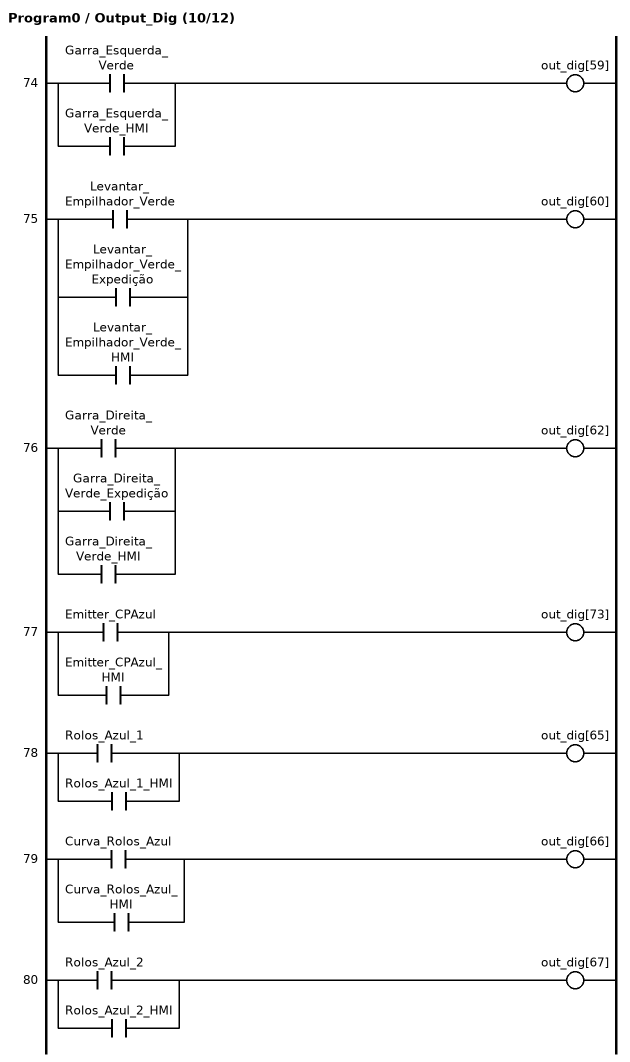
(* [picture p24: Program0 / Output_Dig, rungs 74-80] *)
(* Rung 74 *)
out_dig[59] := Garra_Esquerda_Verde OR Garra_Esquerda_Verde_HMI;
(* Rung 75 *)
out_dig[60] := Levantar_Empilhador_Verde OR Levantar_Empilhador_Verde_Expedição OR Levantar_Empilhador_Verde_HMI;
(* Rung 76 *)
out_dig[62] := Garra_Direita_Verde OR Garra_Direita_Verde_Expedição OR Garra_Direita_Verde_HMI;
(* Rung 77 *)
out_dig[73] := Emitter_CPAzul OR Emitter_CPAzul_HMI;
(* Rung 78 *)
out_dig[65] := Rolos_Azul_1 OR Rolos_Azul_1_HMI;
(* Rung 79 *)
out_dig[66] := Curva_Rolos_Azul OR Curva_Rolos_Azul_HMI;
(* Rung 80 *)
out_dig[67] := Rolos_Azul_2 OR Rolos_Azul_2_HMI;

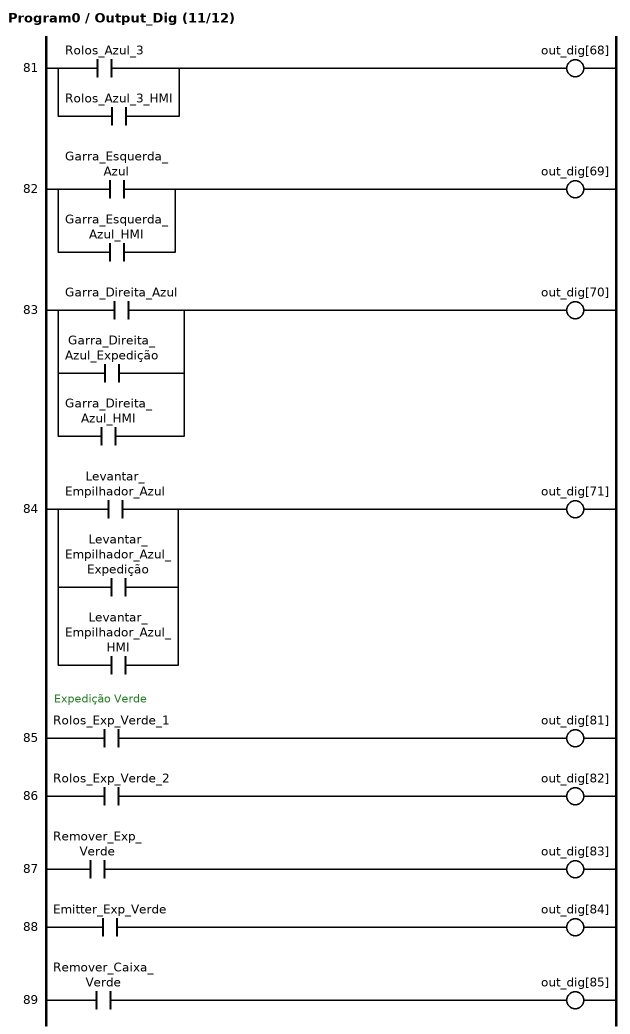
(* Rung 81 *)
out_dig[68] := Rolos_Azul_3 OR Rolos_Azul_3_HMI;
(* Rung 82 *)
out_dig[69] := Garra_Esquerda_Azul OR Garra_Esquerda_Azul_HMI;
(* Rung 83 *)
out_dig[70] := Garra_Direita_Azul OR Garra_Direita_Azul_Expedição OR Garra_Direita_Azul_HMI;
(* Rung 84 *)
out_dig[71] := Levantar_Empilhador_Azul OR Levantar_Empilhador_Azul_Expedição OR Levantar_Empilhador_Azul_HMI;
(* Rung 85: Expedição Verde *)
out_dig[81] := Rolos_Exp_Verde_1;
(* Rung 86 *)
out_dig[82] := Rolos_Exp_Verde_2;
(* Rung 87 *)
out_dig[83] := Remover_Exp_Verde;
(* Rung 88 *)
out_dig[84] := Emitter_Exp_Verde;
(* Rung 89 *)
out_dig[85] := Remover_Caixa_Verde;

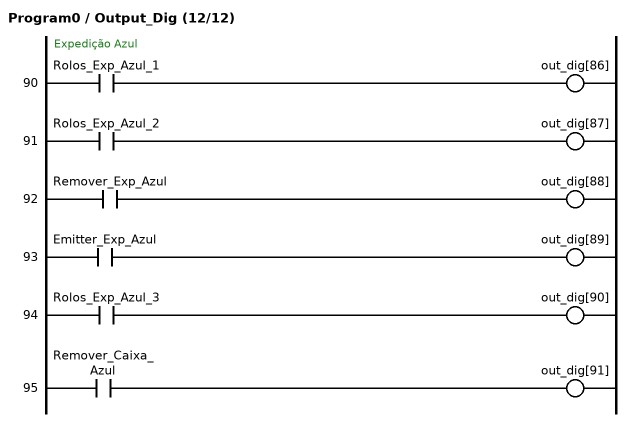
(* Rung 90: Expedição Azul *)
out_dig[86] := Rolos_Exp_Azul_1;
(* Rung 91 *)
out_dig[87] := Rolos_Exp_Azul_2;
(* Rung 92 *)
out_dig[88] := Remover_Exp_Azul;
(* Rung 93 *)
out_dig[89] := Emitter_Exp_Azul;
(* Rung 94 *)
out_dig[90] := Rolos_Exp_Azul_3;
(* Rung 95 *)
out_dig[91] := Remover_Caixa_Azul;

(* Section Separação_Inicial_Etapas: ladder, written here as Structured Text *)

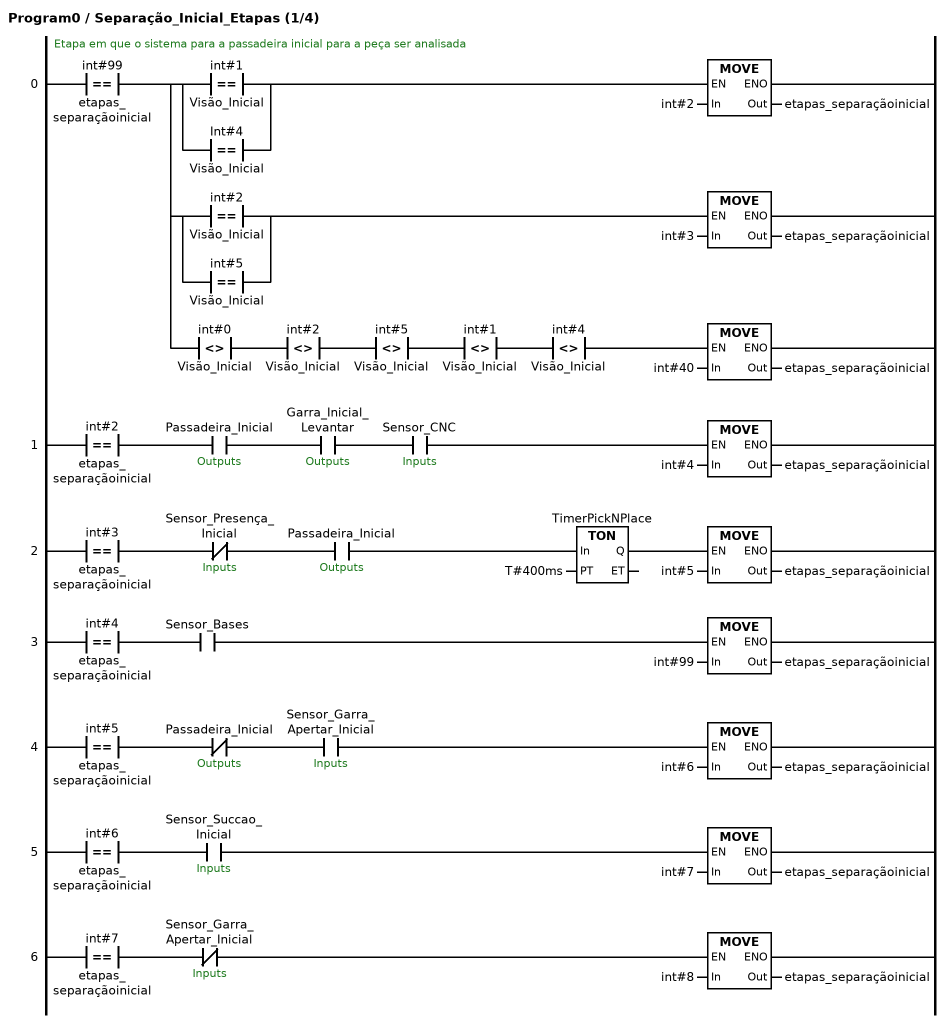
(* Rung 0: Etapa em que o sistema para a passadeira inicial para a peça ser analisada *)
_p4 := int#99 = etapas_separaçãoinicial;
IF (int#99 = etapas_separaçãoinicial) AND ((int#1 = Visão_Inicial) OR (Int#4 = Visão_Inicial)) THEN
    etapas_separaçãoinicial := int#2;
END_IF;
IF _p4 AND ((int#2 = Visão_Inicial) OR (int#5 = Visão_Inicial)) THEN
    etapas_separaçãoinicial := int#3;
END_IF;
IF _p4 AND (int#0 <> Visão_Inicial) AND (int#2 <> Visão_Inicial) AND (int#5 <> Visão_Inicial) AND (int#1 <> Visão_Inicial) AND (int#4 <> Visão_Inicial) THEN
    etapas_separaçãoinicial := int#40;
END_IF;
(* Rung 1 *)
IF (int#2 = etapas_separaçãoinicial) AND Passadeira_Inicial AND Garra_Inicial_Levantar AND Sensor_CNC THEN
    etapas_separaçãoinicial := int#4;
END_IF;
(* Rung 2 *)
TimerPickNPlace(In := (int#3 = etapas_separaçãoinicial) AND NOT Sensor_Presença_Inicial AND Passadeira_Inicial, PT := T#400ms);
IF TimerPickNPlace.Q THEN etapas_separaçãoinicial := int#5; END_IF;
(* Rung 3 *)
IF (int#4 = etapas_separaçãoinicial) AND Sensor_Bases THEN etapas_separaçãoinicial := int#99; END_IF;
(* Rung 4 *)
IF (int#5 = etapas_separaçãoinicial) AND NOT Passadeira_Inicial AND Sensor_Garra_Apertar_Inicial THEN
    etapas_separaçãoinicial := int#6;
END_IF;
(* Rung 5 *)
IF (int#6 = etapas_separaçãoinicial) AND Sensor_Succao_Inicial THEN
    etapas_separaçãoinicial := int#7;
END_IF;
(* Rung 6 *)
IF (int#7 = etapas_separaçãoinicial) AND NOT Sensor_Garra_Apertar_Inicial THEN
    etapas_separaçãoinicial := int#8;
END_IF;

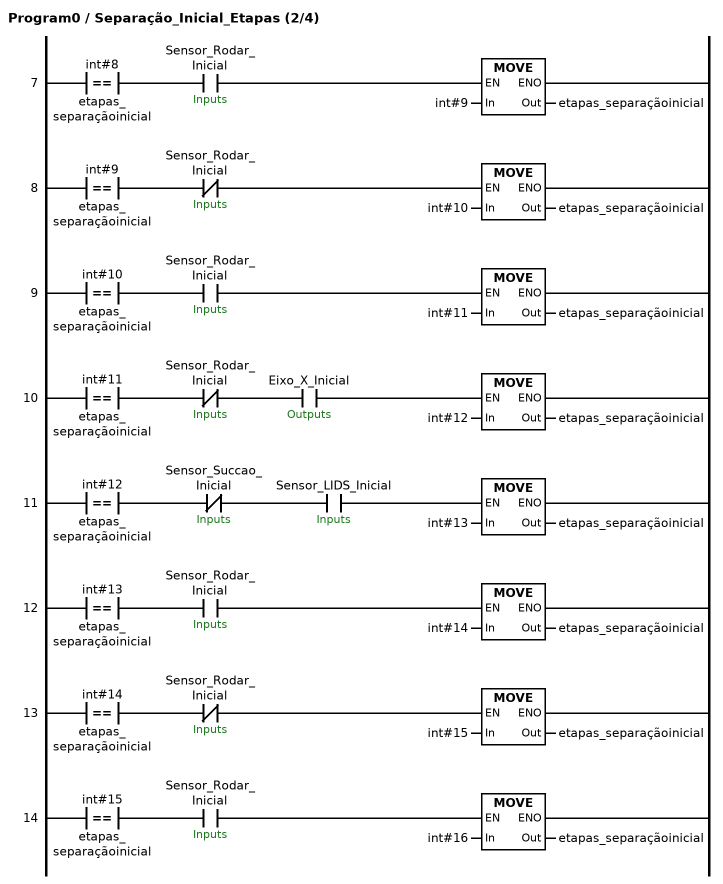
(* Rung 7 *)
IF (int#8 = etapas_separaçãoinicial) AND Sensor_Rodar_Inicial THEN
    etapas_separaçãoinicial := int#9;
END_IF;
(* Rung 8 *)
IF (int#9 = etapas_separaçãoinicial) AND NOT Sensor_Rodar_Inicial THEN
    etapas_separaçãoinicial := int#10;
END_IF;
(* Rung 9 *)
IF (int#10 = etapas_separaçãoinicial) AND Sensor_Rodar_Inicial THEN
    etapas_separaçãoinicial := int#11;
END_IF;
(* Rung 10 *)
IF (int#11 = etapas_separaçãoinicial) AND NOT Sensor_Rodar_Inicial AND Eixo_X_Inicial THEN
    etapas_separaçãoinicial := int#12;
END_IF;
(* Rung 11 *)
IF (int#12 = etapas_separaçãoinicial) AND NOT Sensor_Succao_Inicial AND Sensor_LIDS_Inicial THEN
    etapas_separaçãoinicial := int#13;
END_IF;
(* Rung 12 *)
IF (int#13 = etapas_separaçãoinicial) AND Sensor_Rodar_Inicial THEN
    etapas_separaçãoinicial := int#14;
END_IF;
(* Rung 13 *)
IF (int#14 = etapas_separaçãoinicial) AND NOT Sensor_Rodar_Inicial THEN
    etapas_separaçãoinicial := int#15;
END_IF;
(* Rung 14 *)
IF (int#15 = etapas_separaçãoinicial) AND Sensor_Rodar_Inicial THEN
    etapas_separaçãoinicial := int#16;
END_IF;

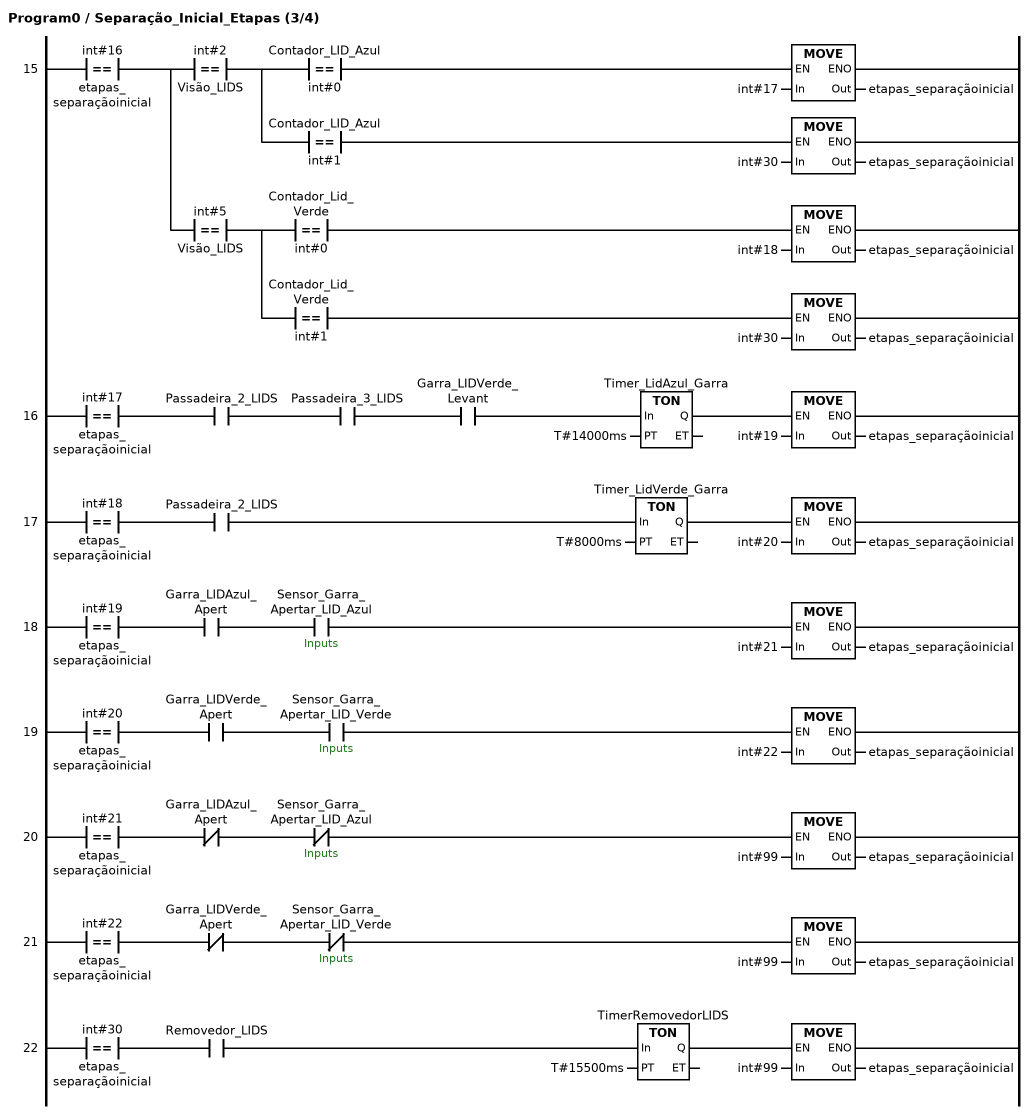
(* Rung 15 *)
_p5 := (int#16 = etapas_separaçãoinicial) AND (int#2 = Visão_LIDS);
_p6 := int#16 = etapas_separaçãoinicial;
IF _p5 AND (Contador_LID_Azul = int#0) THEN etapas_separaçãoinicial := int#17; END_IF;
IF _p5 AND (Contador_LID_Azul = int#1) THEN etapas_separaçãoinicial := int#30; END_IF;
IF _p6 AND (int#5 = Visão_LIDS) AND (Contador_Lid_Verde = int#0) THEN
    etapas_separaçãoinicial := int#18;
END_IF;
IF _p6 AND (int#5 = Visão_LIDS) AND (Contador_Lid_Verde = int#1) THEN
    etapas_separaçãoinicial := int#30;
END_IF;
(* Rung 16 *)
Timer_LidAzul_Garra(In := (int#17 = etapas_separaçãoinicial) AND Passadeira_2_LIDS AND Passadeira_3_LIDS AND Garra_LIDVerde_Levant, PT := T#14000ms);
IF Timer_LidAzul_Garra.Q THEN etapas_separaçãoinicial := int#19; END_IF;
(* Rung 17 *)
Timer_LidVerde_Garra(In := (int#18 = etapas_separaçãoinicial) AND Passadeira_2_LIDS, PT := T#8000ms);
IF Timer_LidVerde_Garra.Q THEN etapas_separaçãoinicial := int#20; END_IF;
(* Rung 18 *)
IF (int#19 = etapas_separaçãoinicial) AND Garra_LIDAzul_Apert AND Sensor_Garra_Apertar_LID_Azul THEN
    etapas_separaçãoinicial := int#21;
END_IF;
(* Rung 19 *)
IF (int#20 = etapas_separaçãoinicial) AND Garra_LIDVerde_Apert AND Sensor_Garra_Apertar_LID_Verde THEN
    etapas_separaçãoinicial := int#22;
END_IF;
(* Rung 20 *)
IF (int#21 = etapas_separaçãoinicial) AND NOT Garra_LIDAzul_Apert AND NOT Sensor_Garra_Apertar_LID_Azul THEN
    etapas_separaçãoinicial := int#99;
END_IF;
(* Rung 21 *)
IF (int#22 = etapas_separaçãoinicial) AND NOT Garra_LIDVerde_Apert AND NOT Sensor_Garra_Apertar_LID_Verde THEN
    etapas_separaçãoinicial := int#99;
END_IF;
(* Rung 22 *)
TimerRemovedorLIDS(In := (int#30 = etapas_separaçãoinicial) AND Removedor_LIDS, PT := T#15500ms);
IF TimerRemovedorLIDS.Q THEN etapas_separaçãoinicial := int#99; END_IF;

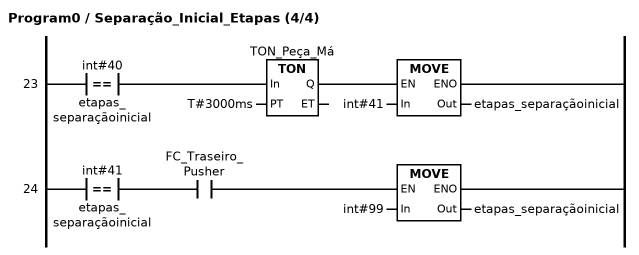
(* Rung 23 *)
TON_Peça_Má(In := int#40 = etapas_separaçãoinicial, PT := T#3000ms);
IF TON_Peça_Má.Q THEN etapas_separaçãoinicial := int#41; END_IF;
(* Rung 24 *)
IF (int#41 = etapas_separaçãoinicial) AND FC_Traseiro_Pusher THEN
    etapas_separaçãoinicial := int#99;
END_IF;

(* Section Separação_Inicial_Saídas: ladder, written here as Structured Text *)

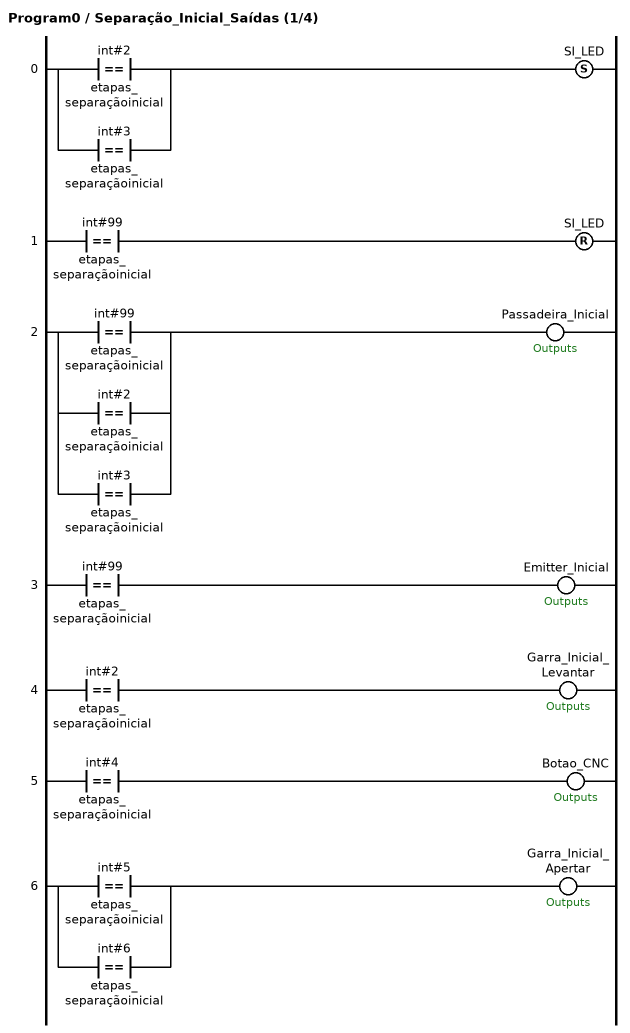
(* Rung 0 *)
IF (int#2 = etapas_separaçãoinicial) OR (int#3 = etapas_separaçãoinicial) THEN SI_LED := TRUE; END_IF;
(* Rung 1 *)
IF int#99 = etapas_separaçãoinicial THEN SI_LED := FALSE; END_IF;
(* Rung 2 *)
Passadeira_Inicial := (int#99 = etapas_separaçãoinicial) OR (int#2 = etapas_separaçãoinicial) OR (int#3 = etapas_separaçãoinicial);
(* Rung 3 *)
Emitter_Inicial := int#99 = etapas_separaçãoinicial;
(* Rung 4 *)
Garra_Inicial_Levantar := int#2 = etapas_separaçãoinicial;
(* Rung 5 *)
Botao_CNC := int#4 = etapas_separaçãoinicial;
(* Rung 6 *)
Garra_Inicial_Apertar := (int#5 = etapas_separaçãoinicial) OR (int#6 = etapas_separaçãoinicial);

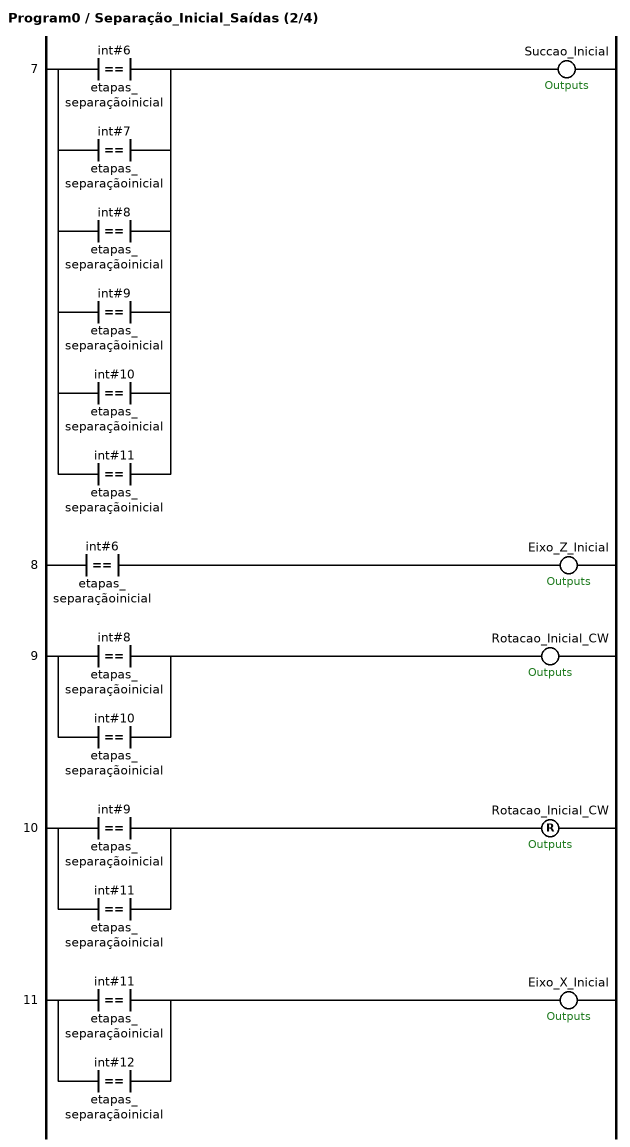
(* Rung 7 *)
Succao_Inicial := (int#6 = etapas_separaçãoinicial) OR (int#7 = etapas_separaçãoinicial) OR (int#8 = etapas_separaçãoinicial) OR (int#9 = etapas_separaçãoinicial) OR (int#10 = etapas_separaçãoinicial) OR (int#11 = etapas_separaçãoinicial);
(* Rung 8 *)
Eixo_Z_Inicial := int#6 = etapas_separaçãoinicial;
(* Rung 9 *)
Rotacao_Inicial_CW := (int#8 = etapas_separaçãoinicial) OR (int#10 = etapas_separaçãoinicial);
(* Rung 10 *)
IF (int#9 = etapas_separaçãoinicial) OR (int#11 = etapas_separaçãoinicial) THEN
    Rotacao_Inicial_CW := FALSE;
END_IF;
(* Rung 11 *)
Eixo_X_Inicial := (int#11 = etapas_separaçãoinicial) OR (int#12 = etapas_separaçãoinicial);

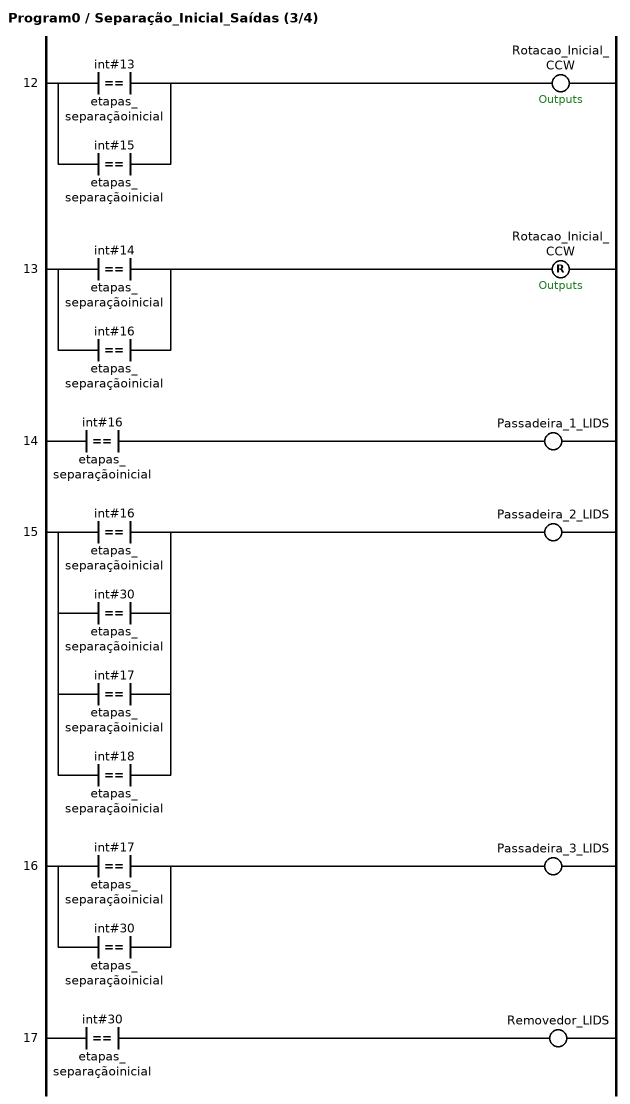
(* Rung 12 *)
Rotacao_Inicial_CCW := (int#13 = etapas_separaçãoinicial) OR (int#15 = etapas_separaçãoinicial);
(* Rung 13 *)
IF (int#14 = etapas_separaçãoinicial) OR (int#16 = etapas_separaçãoinicial) THEN
    Rotacao_Inicial_CCW := FALSE;
END_IF;
(* Rung 14 *)
Passadeira_1_LIDS := int#16 = etapas_separaçãoinicial;
(* Rung 15 *)
Passadeira_2_LIDS := (int#16 = etapas_separaçãoinicial) OR (int#30 = etapas_separaçãoinicial) OR (int#17 = etapas_separaçãoinicial) OR (int#18 = etapas_separaçãoinicial);
(* Rung 16 *)
Passadeira_3_LIDS := (int#17 = etapas_separaçãoinicial) OR (int#30 = etapas_separaçãoinicial);
(* Rung 17 *)
Removedor_LIDS := int#30 = etapas_separaçãoinicial;

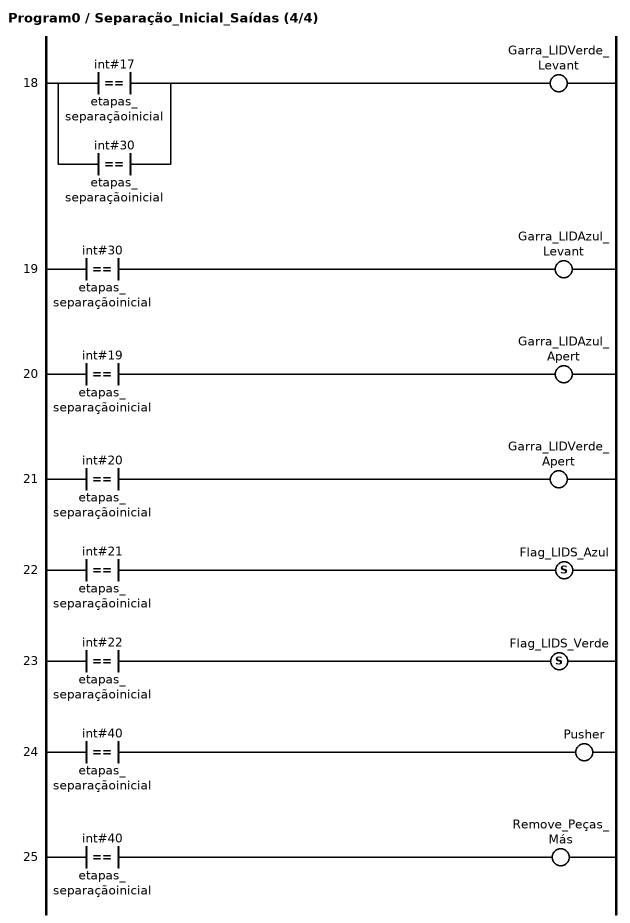
(* Rung 18 *)
Garra_LIDVerde_Levant := (int#17 = etapas_separaçãoinicial) OR (int#30 = etapas_separaçãoinicial);
(* Rung 19 *)
Garra_LIDAzul_Levant := int#30 = etapas_separaçãoinicial;
(* Rung 20 *)
Garra_LIDAzul_Apert := int#19 = etapas_separaçãoinicial;
(* Rung 21 *)
Garra_LIDVerde_Apert := int#20 = etapas_separaçãoinicial;
(* Rung 22 *)
IF int#21 = etapas_separaçãoinicial THEN Flag_LIDS_Azul := TRUE; END_IF;
(* Rung 23 *)
IF int#22 = etapas_separaçãoinicial THEN Flag_LIDS_Verde := TRUE; END_IF;
(* Rung 24 *)
Pusher := int#40 = etapas_separaçãoinicial;
(* Rung 25 *)
Remove_Peças_Más := int#40 = etapas_separaçãoinicial;

(* Section Bases_Etapas: ladder, written here as Structured Text *)

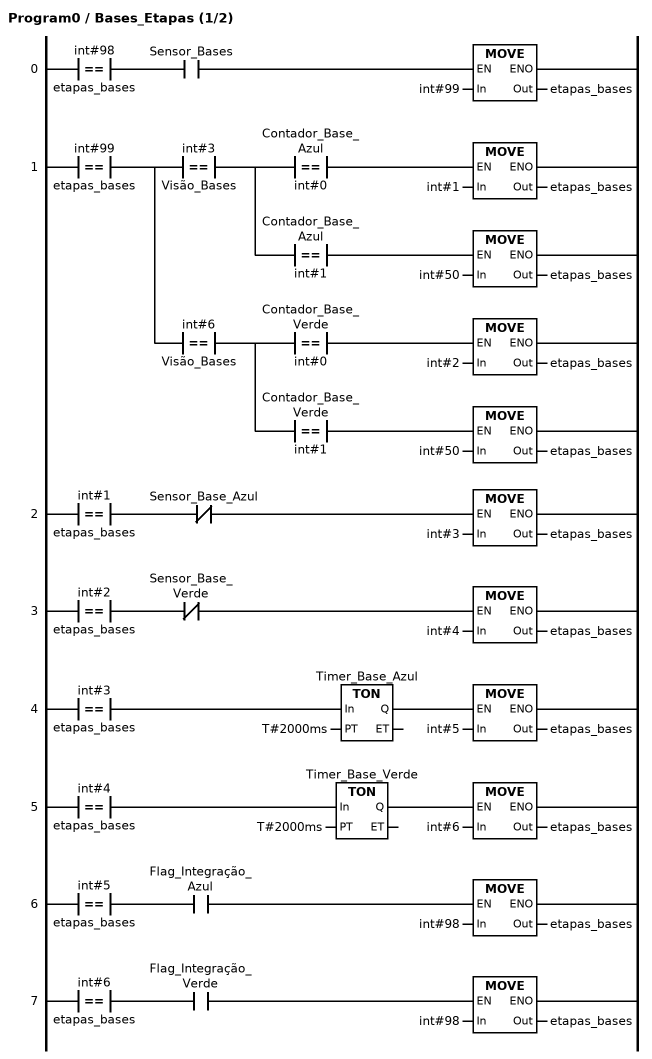
(* Rung 0 *)
IF (int#98 = etapas_bases) AND Sensor_Bases THEN etapas_bases := int#99; END_IF;
(* Rung 1 *)
_p7 := (int#99 = etapas_bases) AND (int#3 = Visão_Bases);
_p8 := int#99 = etapas_bases;
IF _p7 AND (Contador_Base_Azul = int#0) THEN etapas_bases := int#1; END_IF;
IF _p7 AND (Contador_Base_Azul = int#1) THEN etapas_bases := int#50; END_IF;
IF _p8 AND (int#6 = Visão_Bases) AND (Contador_Base_Verde = int#0) THEN etapas_bases := int#2; END_IF;
IF _p8 AND (int#6 = Visão_Bases) AND (Contador_Base_Verde = int#1) THEN etapas_bases := int#50; END_IF;
(* Rung 2 *)
IF (int#1 = etapas_bases) AND NOT Sensor_Base_Azul THEN etapas_bases := int#3; END_IF;
(* Rung 3 *)
IF (int#2 = etapas_bases) AND NOT Sensor_Base_Verde THEN etapas_bases := int#4; END_IF;
(* Rung 4 *)
Timer_Base_Azul(In := int#3 = etapas_bases, PT := T#2000ms);
IF Timer_Base_Azul.Q THEN etapas_bases := int#5; END_IF;
(* Rung 5 *)
Timer_Base_Verde(In := int#4 = etapas_bases, PT := T#2000ms);
IF Timer_Base_Verde.Q THEN etapas_bases := int#6; END_IF;
(* Rung 6 *)
IF (int#5 = etapas_bases) AND Flag_Integração_Azul THEN etapas_bases := int#98; END_IF;
(* Rung 7 *)
IF (int#6 = etapas_bases) AND Flag_Integração_Verde THEN etapas_bases := int#98; END_IF;

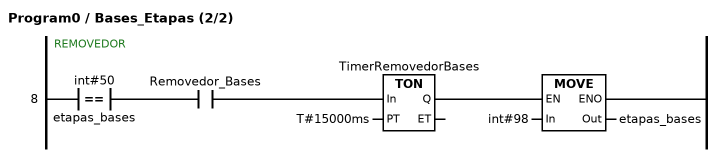
(* Rung 8: REMOVEDOR *)
TimerRemovedorBases(In := (int#50 = etapas_bases) AND Removedor_Bases, PT := T#15000ms);
IF TimerRemovedorBases.Q THEN etapas_bases := int#98; END_IF;

(* Section Bases_Saídas: ladder, written here as Structured Text *)

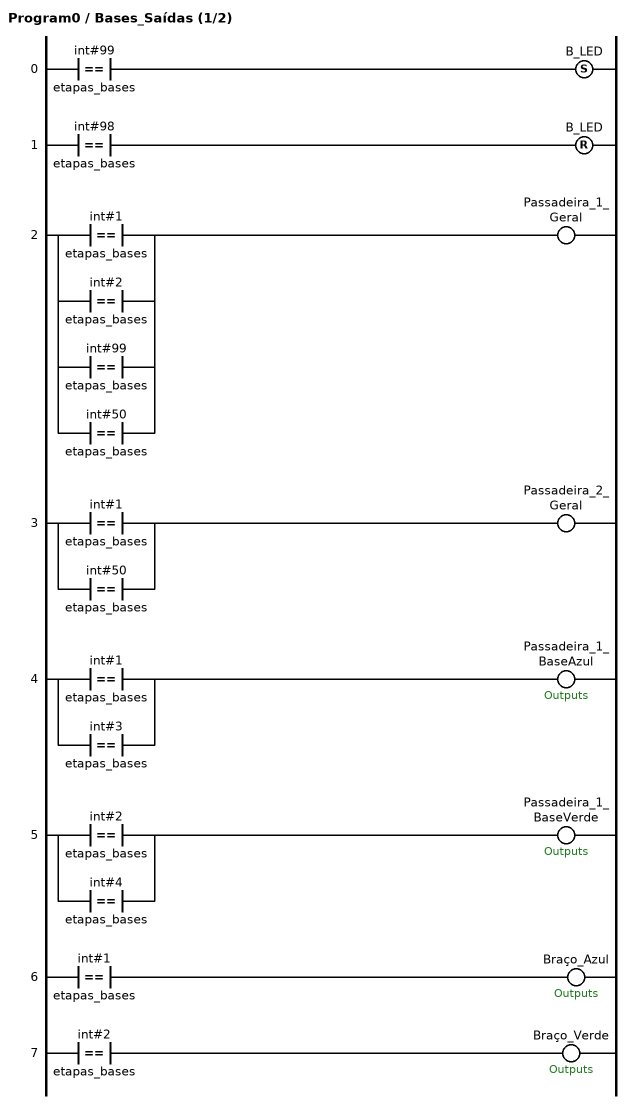
(* Rung 0 *)
IF int#99 = etapas_bases THEN B_LED := TRUE; END_IF;
(* Rung 1 *)
IF int#98 = etapas_bases THEN B_LED := FALSE; END_IF;
(* Rung 2 *)
Passadeira_1_Geral := (int#1 = etapas_bases) OR (int#2 = etapas_bases) OR (int#99 = etapas_bases) OR (int#50 = etapas_bases);
(* Rung 3 *)
Passadeira_2_Geral := (int#1 = etapas_bases) OR (int#50 = etapas_bases);
(* Rung 4 *)
Passadeira_1_BaseAzul := (int#1 = etapas_bases) OR (int#3 = etapas_bases);
(* Rung 5 *)
Passadeira_1_BaseVerde := (int#2 = etapas_bases) OR (int#4 = etapas_bases);
(* Rung 6 *)
Braço_Azul := int#1 = etapas_bases;
(* Rung 7 *)
Braço_Verde := int#2 = etapas_bases;

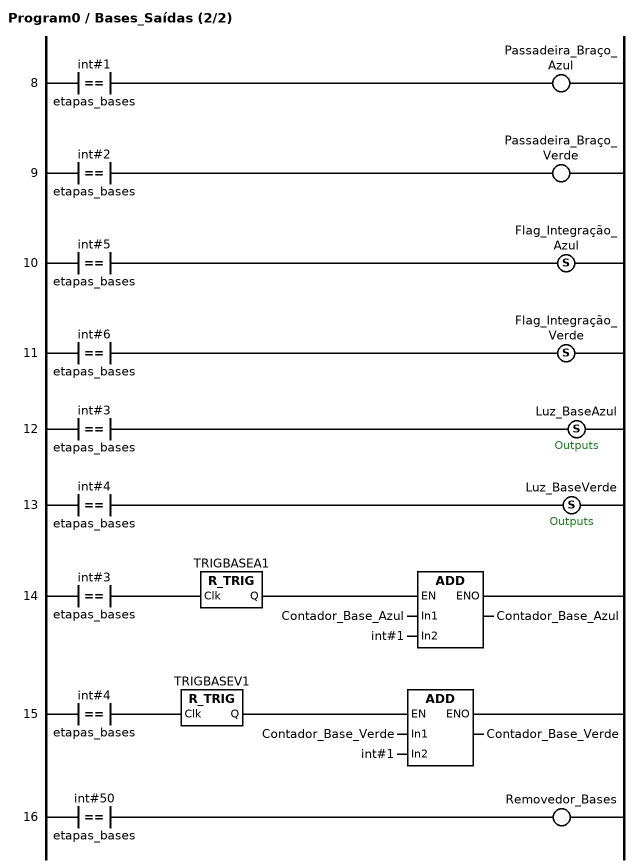
(* Rung 8 *)
Passadeira_Braço_Azul := int#1 = etapas_bases;
(* Rung 9 *)
Passadeira_Braço_Verde := int#2 = etapas_bases;
(* Rung 10 *)
IF int#5 = etapas_bases THEN Flag_Integração_Azul := TRUE; END_IF;
(* Rung 11 *)
IF int#6 = etapas_bases THEN Flag_Integração_Verde := TRUE; END_IF;
(* Rung 12 *)
IF int#3 = etapas_bases THEN Luz_BaseAzul := TRUE; END_IF;
(* Rung 13 *)
IF int#4 = etapas_bases THEN Luz_BaseVerde := TRUE; END_IF;
(* Rung 14 *)
TRIGBASEA1(Clk := int#3 = etapas_bases);
IF TRIGBASEA1.Q THEN Contador_Base_Azul := Contador_Base_Azul + int#1; END_IF;
(* Rung 15 *)
TRIGBASEV1(Clk := int#4 = etapas_bases);
IF TRIGBASEV1.Q THEN Contador_Base_Verde := Contador_Base_Verde + int#1; END_IF;
(* Rung 16 *)
Removedor_Bases := int#50 = etapas_bases;

(* Section LIDS_Etapas: ladder, written here as Structured Text *)

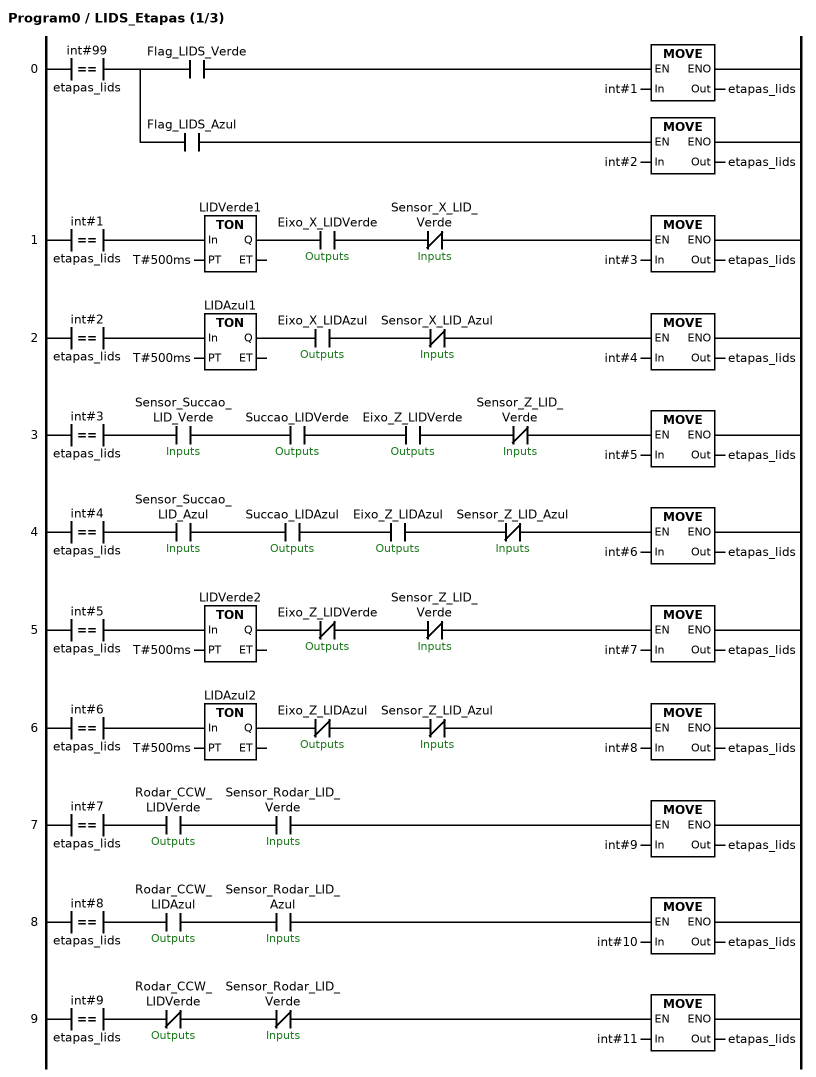
(* Rung 0 *)
_p9 := int#99 = etapas_lids;
IF (int#99 = etapas_lids) AND Flag_LIDS_Verde THEN etapas_lids := int#1; END_IF;
IF _p9 AND Flag_LIDS_Azul THEN etapas_lids := int#2; END_IF;
(* Rung 1 *)
LIDVerde1(In := int#1 = etapas_lids, PT := T#500ms);
IF LIDVerde1.Q AND Eixo_X_LIDVerde AND NOT Sensor_X_LID_Verde THEN etapas_lids := int#3; END_IF;
(* Rung 2 *)
LIDAzul1(In := int#2 = etapas_lids, PT := T#500ms);
IF LIDAzul1.Q AND Eixo_X_LIDAzul AND NOT Sensor_X_LID_Azul THEN etapas_lids := int#4; END_IF;
(* Rung 3 *)
IF (int#3 = etapas_lids) AND Sensor_Succao_LID_Verde AND Succao_LIDVerde AND Eixo_Z_LIDVerde AND NOT Sensor_Z_LID_Verde THEN
    etapas_lids := int#5;
END_IF;
(* Rung 4 *)
IF (int#4 = etapas_lids) AND Sensor_Succao_LID_Azul AND Succao_LIDAzul AND Eixo_Z_LIDAzul AND NOT Sensor_Z_LID_Azul THEN
    etapas_lids := int#6;
END_IF;
(* Rung 5 *)
LIDVerde2(In := int#5 = etapas_lids, PT := T#500ms);
IF LIDVerde2.Q AND NOT Eixo_Z_LIDVerde AND NOT Sensor_Z_LID_Verde THEN etapas_lids := int#7; END_IF;
(* Rung 6 *)
LIDAzul2(In := int#6 = etapas_lids, PT := T#500ms);
IF LIDAzul2.Q AND NOT Eixo_Z_LIDAzul AND NOT Sensor_Z_LID_Azul THEN etapas_lids := int#8; END_IF;
(* Rung 7 *)
IF (int#7 = etapas_lids) AND Rodar_CCW_LIDVerde AND Sensor_Rodar_LID_Verde THEN
    etapas_lids := int#9;
END_IF;
(* Rung 8 *)
IF (int#8 = etapas_lids) AND Rodar_CCW_LIDAzul AND Sensor_Rodar_LID_Azul THEN
    etapas_lids := int#10;
END_IF;
(* Rung 9 *)
IF (int#9 = etapas_lids) AND NOT Rodar_CCW_LIDVerde AND NOT Sensor_Rodar_LID_Verde THEN
    etapas_lids := int#11;
END_IF;

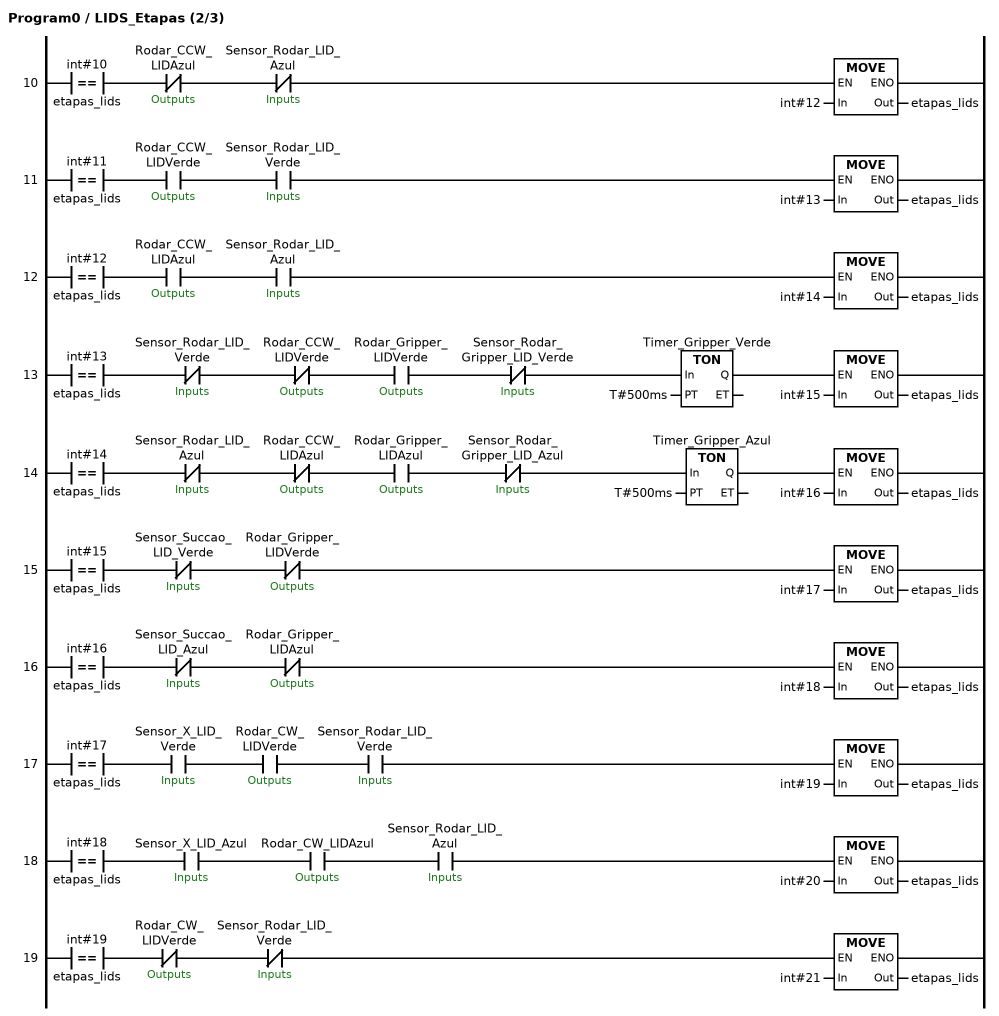
(* Rung 10 *)
IF (int#10 = etapas_lids) AND NOT Rodar_CCW_LIDAzul AND NOT Sensor_Rodar_LID_Azul THEN
    etapas_lids := int#12;
END_IF;
(* Rung 11 *)
IF (int#11 = etapas_lids) AND Rodar_CCW_LIDVerde AND Sensor_Rodar_LID_Verde THEN
    etapas_lids := int#13;
END_IF;
(* Rung 12 *)
IF (int#12 = etapas_lids) AND Rodar_CCW_LIDAzul AND Sensor_Rodar_LID_Azul THEN
    etapas_lids := int#14;
END_IF;
(* Rung 13 *)
Timer_Gripper_Verde(In := (int#13 = etapas_lids) AND NOT Sensor_Rodar_LID_Verde AND NOT Rodar_CCW_LIDVerde AND Rodar_Gripper_LIDVerde AND NOT Sensor_Rodar_Gripper_LID_Verde, PT := T#500ms);
IF Timer_Gripper_Verde.Q THEN etapas_lids := int#15; END_IF;
(* Rung 14 *)
Timer_Gripper_Azul(In := (int#14 = etapas_lids) AND NOT Sensor_Rodar_LID_Azul AND NOT Rodar_CCW_LIDAzul AND Rodar_Gripper_LIDAzul AND NOT Sensor_Rodar_Gripper_LID_Azul, PT := T#500ms);
IF Timer_Gripper_Azul.Q THEN etapas_lids := int#16; END_IF;
(* Rung 15 *)
IF (int#15 = etapas_lids) AND NOT Sensor_Succao_LID_Verde AND NOT Rodar_Gripper_LIDVerde THEN
    etapas_lids := int#17;
END_IF;
(* Rung 16 *)
IF (int#16 = etapas_lids) AND NOT Sensor_Succao_LID_Azul AND NOT Rodar_Gripper_LIDAzul THEN
    etapas_lids := int#18;
END_IF;
(* Rung 17 *)
IF (int#17 = etapas_lids) AND Sensor_X_LID_Verde AND Rodar_CW_LIDVerde AND Sensor_Rodar_LID_Verde THEN
    etapas_lids := int#19;
END_IF;
(* Rung 18 *)
IF (int#18 = etapas_lids) AND Sensor_X_LID_Azul AND Rodar_CW_LIDAzul AND Sensor_Rodar_LID_Azul THEN
    etapas_lids := int#20;
END_IF;
(* Rung 19 *)
IF (int#19 = etapas_lids) AND NOT Rodar_CW_LIDVerde AND NOT Sensor_Rodar_LID_Verde THEN
    etapas_lids := int#21;
END_IF;

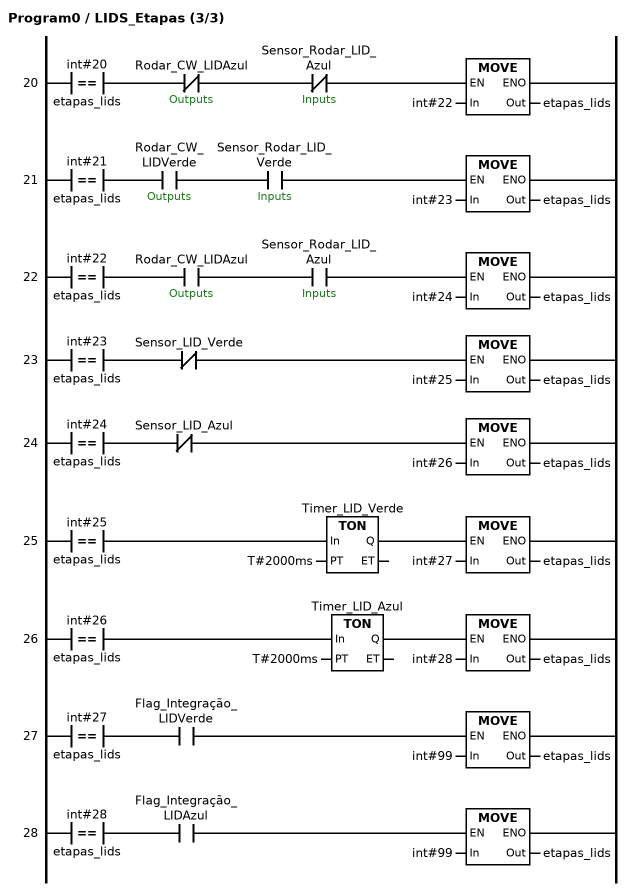
(* Rung 20 *)
IF (int#20 = etapas_lids) AND NOT Rodar_CW_LIDAzul AND NOT Sensor_Rodar_LID_Azul THEN
    etapas_lids := int#22;
END_IF;
(* Rung 21 *)
IF (int#21 = etapas_lids) AND Rodar_CW_LIDVerde AND Sensor_Rodar_LID_Verde THEN
    etapas_lids := int#23;
END_IF;
(* Rung 22 *)
IF (int#22 = etapas_lids) AND Rodar_CW_LIDAzul AND Sensor_Rodar_LID_Azul THEN
    etapas_lids := int#24;
END_IF;
(* Rung 23 *)
IF (int#23 = etapas_lids) AND NOT Sensor_LID_Verde THEN etapas_lids := int#25; END_IF;
(* Rung 24 *)
IF (int#24 = etapas_lids) AND NOT Sensor_LID_Azul THEN etapas_lids := int#26; END_IF;
(* Rung 25 *)
Timer_LID_Verde(In := int#25 = etapas_lids, PT := T#2000ms);
IF Timer_LID_Verde.Q THEN etapas_lids := int#27; END_IF;
(* Rung 26 *)
Timer_LID_Azul(In := int#26 = etapas_lids, PT := T#2000ms);
IF Timer_LID_Azul.Q THEN etapas_lids := int#28; END_IF;
(* Rung 27 *)
IF (int#27 = etapas_lids) AND Flag_Integração_LIDVerde THEN etapas_lids := int#99; END_IF;
(* Rung 28 *)
IF (int#28 = etapas_lids) AND Flag_Integração_LIDAzul THEN etapas_lids := int#99; END_IF;

(* Section LIDS_Saídas: ladder, written here as Structured Text *)

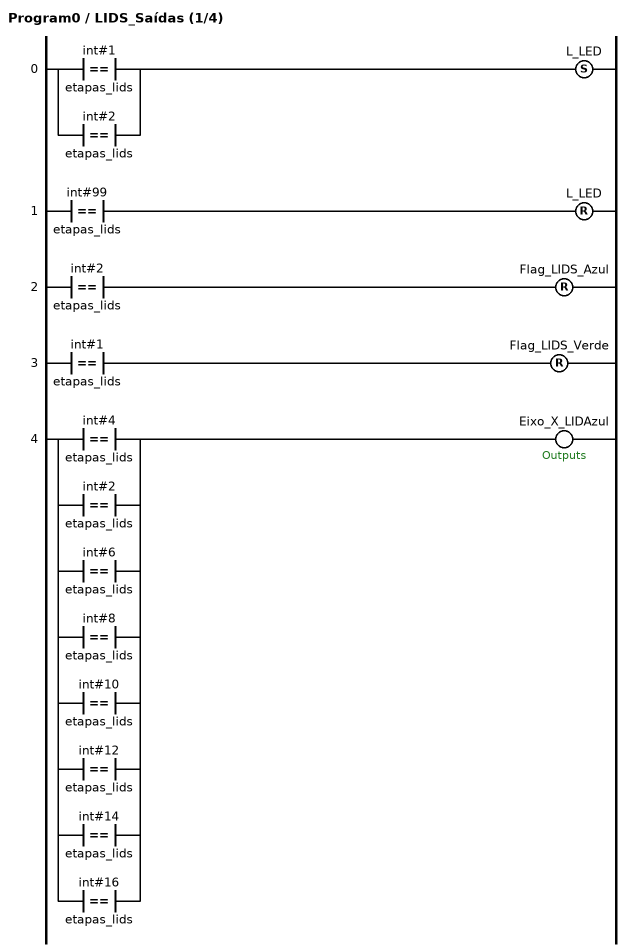
(* Rung 0 *)
IF (int#1 = etapas_lids) OR (int#2 = etapas_lids) THEN L_LED := TRUE; END_IF;
(* Rung 1 *)
IF int#99 = etapas_lids THEN L_LED := FALSE; END_IF;
(* Rung 2 *)
IF int#2 = etapas_lids THEN Flag_LIDS_Azul := FALSE; END_IF;
(* Rung 3 *)
IF int#1 = etapas_lids THEN Flag_LIDS_Verde := FALSE; END_IF;
(* Rung 4 *)
Eixo_X_LIDAzul := (int#4 = etapas_lids) OR (int#2 = etapas_lids) OR (int#6 = etapas_lids) OR (int#8 = etapas_lids) OR (int#10 = etapas_lids) OR (int#12 = etapas_lids) OR (int#14 = etapas_lids) OR (int#16 = etapas_lids);

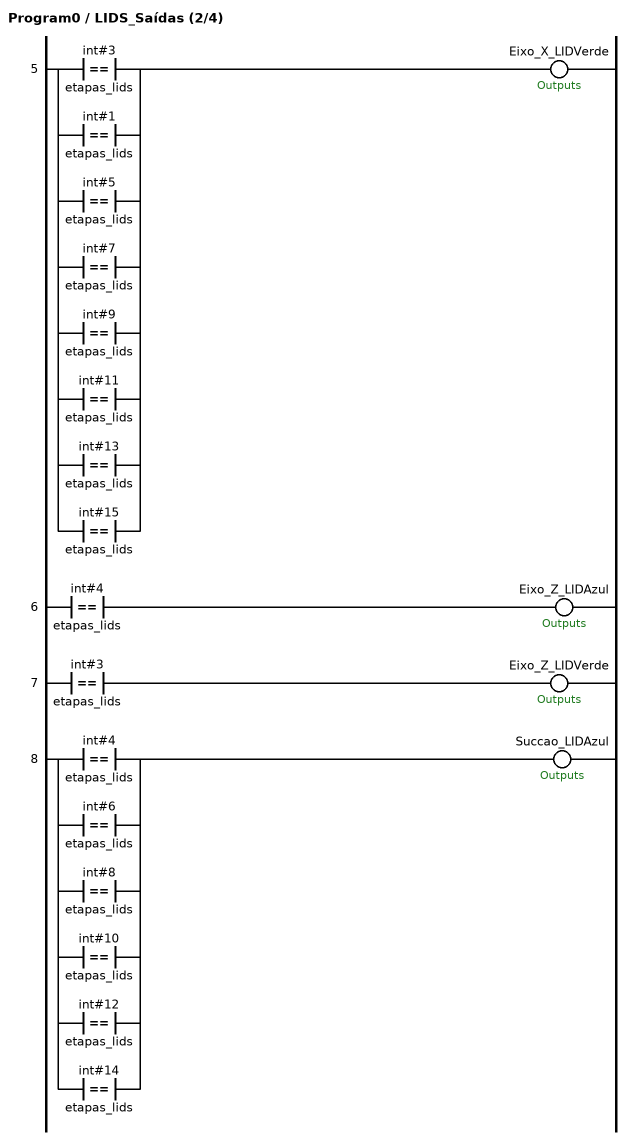
(* Rung 5 *)
Eixo_X_LIDVerde := (int#3 = etapas_lids) OR (int#1 = etapas_lids) OR (int#5 = etapas_lids) OR (int#7 = etapas_lids) OR (int#9 = etapas_lids) OR (int#11 = etapas_lids) OR (int#13 = etapas_lids) OR (int#15 = etapas_lids);
(* Rung 6 *)
Eixo_Z_LIDAzul := int#4 = etapas_lids;
(* Rung 7 *)
Eixo_Z_LIDVerde := int#3 = etapas_lids;
(* Rung 8 *)
Succao_LIDAzul := (int#4 = etapas_lids) OR (int#6 = etapas_lids) OR (int#8 = etapas_lids) OR (int#10 = etapas_lids) OR (int#12 = etapas_lids) OR (int#14 = etapas_lids);

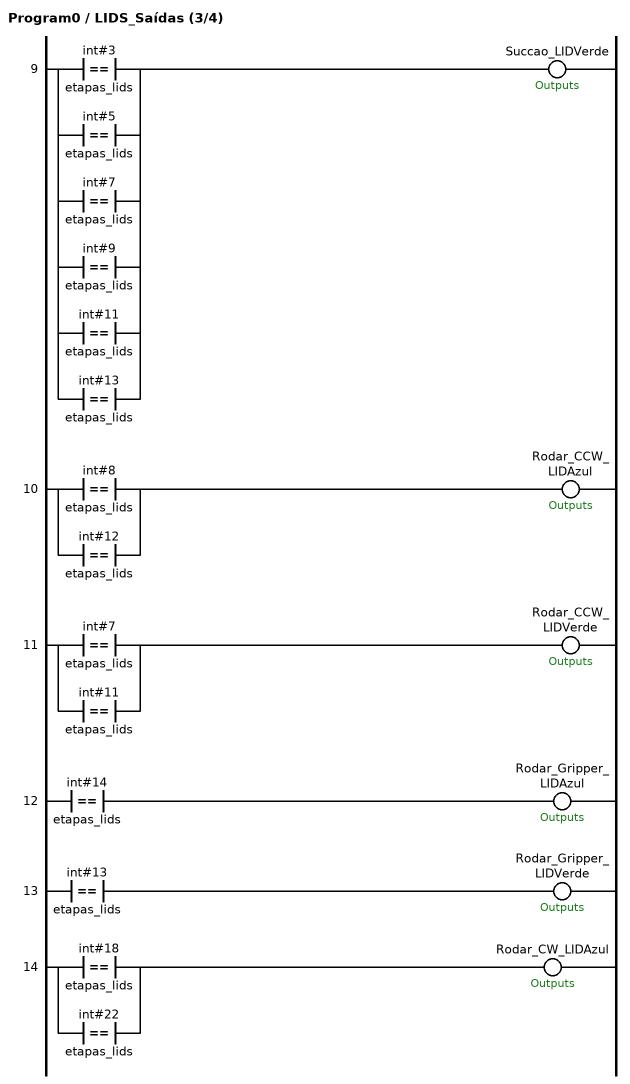
(* Rung 9 *)
Succao_LIDVerde := (int#3 = etapas_lids) OR (int#5 = etapas_lids) OR (int#7 = etapas_lids) OR (int#9 = etapas_lids) OR (int#11 = etapas_lids) OR (int#13 = etapas_lids);
(* Rung 10 *)
Rodar_CCW_LIDAzul := (int#8 = etapas_lids) OR (int#12 = etapas_lids);
(* Rung 11 *)
Rodar_CCW_LIDVerde := (int#7 = etapas_lids) OR (int#11 = etapas_lids);
(* Rung 12 *)
Rodar_Gripper_LIDAzul := int#14 = etapas_lids;
(* Rung 13 *)
Rodar_Gripper_LIDVerde := int#13 = etapas_lids;
(* Rung 14 *)
Rodar_CW_LIDAzul := (int#18 = etapas_lids) OR (int#22 = etapas_lids);

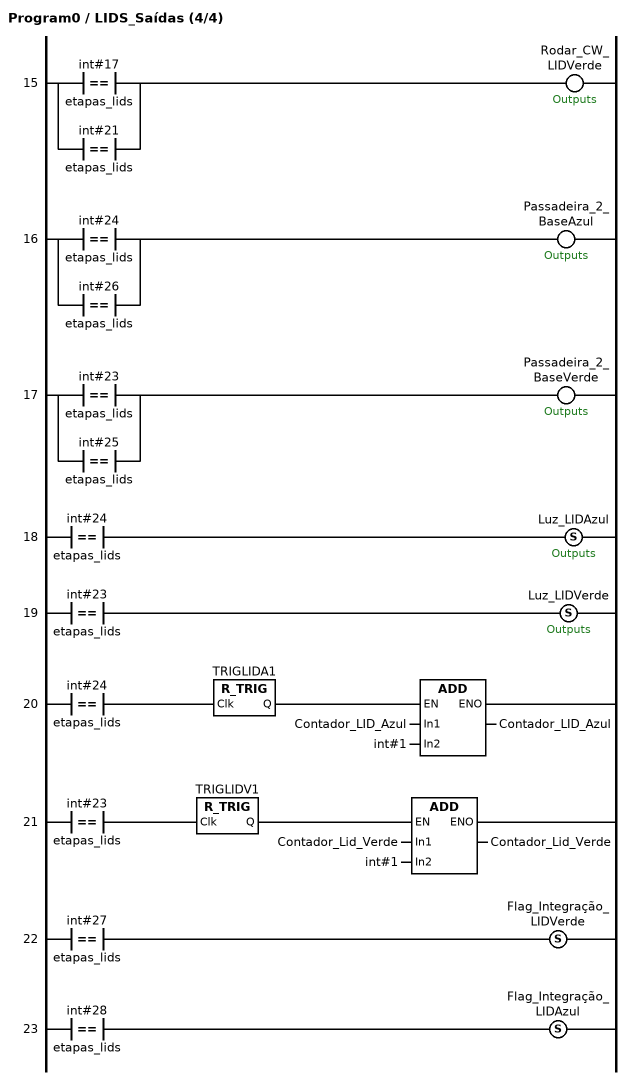
(* Rung 15 *)
Rodar_CW_LIDVerde := (int#17 = etapas_lids) OR (int#21 = etapas_lids);
(* Rung 16 *)
Passadeira_2_BaseAzul := (int#24 = etapas_lids) OR (int#26 = etapas_lids);
(* Rung 17 *)
Passadeira_2_BaseVerde := (int#23 = etapas_lids) OR (int#25 = etapas_lids);
(* Rung 18 *)
IF int#24 = etapas_lids THEN Luz_LIDAzul := TRUE; END_IF;
(* Rung 19 *)
IF int#23 = etapas_lids THEN Luz_LIDVerde := TRUE; END_IF;
(* Rung 20 *)
TRIGLIDA1(Clk := int#24 = etapas_lids);
IF TRIGLIDA1.Q THEN Contador_LID_Azul := Contador_LID_Azul + int#1; END_IF;
(* Rung 21 *)
TRIGLIDV1(Clk := int#23 = etapas_lids);
IF TRIGLIDV1.Q THEN Contador_Lid_Verde := Contador_Lid_Verde + int#1; END_IF;
(* Rung 22 *)
IF int#27 = etapas_lids THEN Flag_Integração_LIDVerde := TRUE; END_IF;
(* Rung 23 *)
IF int#28 = etapas_lids THEN Flag_Integração_LIDAzul := TRUE; END_IF;

(* Section Integração_Etapas: ladder, written here as Structured Text *)

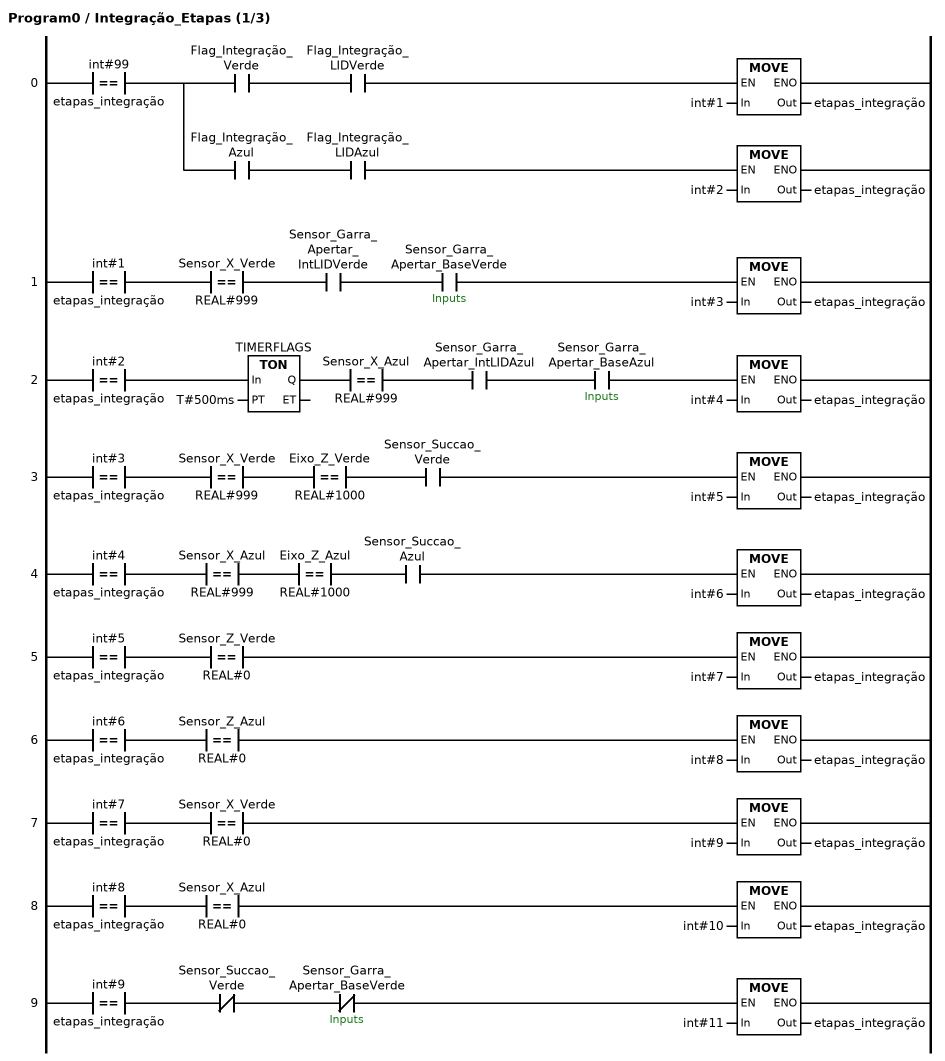
(* Rung 0 *)
_p10 := int#99 = etapas_integração;
IF (int#99 = etapas_integração) AND Flag_Integração_Verde AND Flag_Integração_LIDVerde THEN
    etapas_integração := int#1;
END_IF;
IF _p10 AND Flag_Integração_Azul AND Flag_Integração_LIDAzul THEN etapas_integração := int#2; END_IF;
(* Rung 1 *)
IF (int#1 = etapas_integração) AND (Sensor_X_Verde = REAL#999) AND Sensor_Garra_Apertar_IntLIDVerde AND Sensor_Garra_Apertar_BaseVerde THEN
    etapas_integração := int#3;
END_IF;
(* Rung 2 *)
TIMERFLAGS(In := int#2 = etapas_integração, PT := T#500ms);
IF TIMERFLAGS.Q AND (Sensor_X_Azul = REAL#999) AND Sensor_Garra_Apertar_IntLIDAzul AND Sensor_Garra_Apertar_BaseAzul THEN
    etapas_integração := int#4;
END_IF;
(* Rung 3 *)
IF (int#3 = etapas_integração) AND (Sensor_X_Verde = REAL#999) AND (Eixo_Z_Verde = REAL#1000) AND Sensor_Succao_Verde THEN
    etapas_integração := int#5;
END_IF;
(* Rung 4 *)
IF (int#4 = etapas_integração) AND (Sensor_X_Azul = REAL#999) AND (Eixo_Z_Azul = REAL#1000) AND Sensor_Succao_Azul THEN
    etapas_integração := int#6;
END_IF;
(* Rung 5 *)
IF (int#5 = etapas_integração) AND (Sensor_Z_Verde = REAL#0) THEN etapas_integração := int#7; END_IF;
(* Rung 6 *)
IF (int#6 = etapas_integração) AND (Sensor_Z_Azul = REAL#0) THEN etapas_integração := int#8; END_IF;
(* Rung 7 *)
IF (int#7 = etapas_integração) AND (Sensor_X_Verde = REAL#0) THEN etapas_integração := int#9; END_IF;
(* Rung 8 *)
IF (int#8 = etapas_integração) AND (Sensor_X_Azul = REAL#0) THEN etapas_integração := int#10; END_IF;
(* Rung 9 *)
IF (int#9 = etapas_integração) AND NOT Sensor_Succao_Verde AND NOT Sensor_Garra_Apertar_BaseVerde THEN
    etapas_integração := int#11;
END_IF;

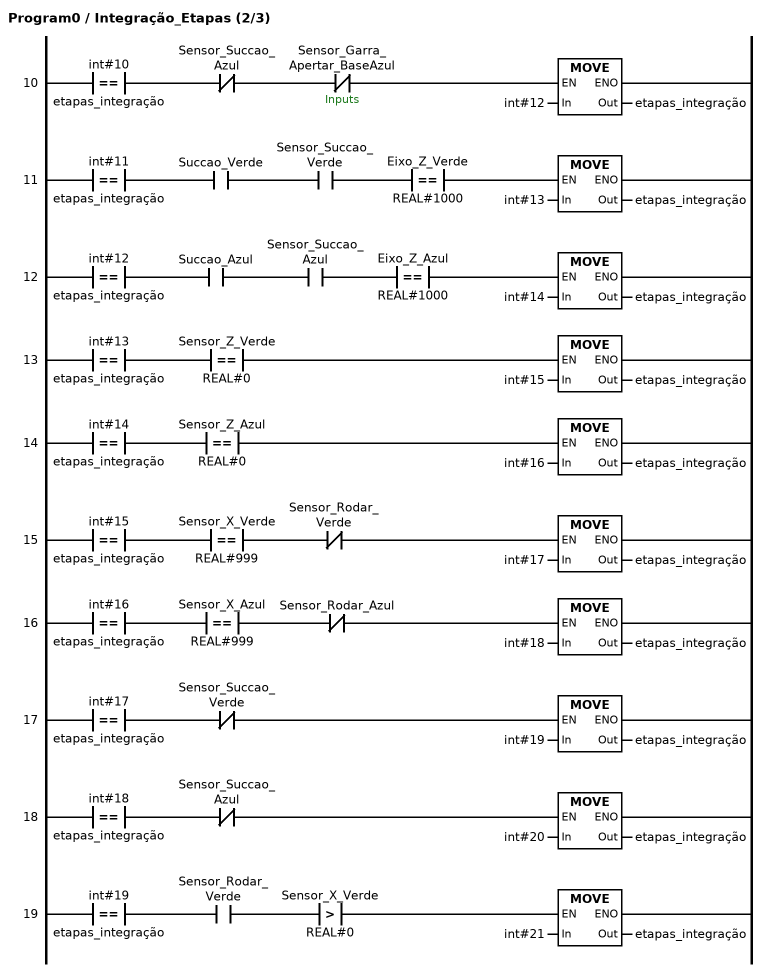
(* Rung 10 *)
IF (int#10 = etapas_integração) AND NOT Sensor_Succao_Azul AND NOT Sensor_Garra_Apertar_BaseAzul THEN
    etapas_integração := int#12;
END_IF;
(* Rung 11 *)
IF (int#11 = etapas_integração) AND Succao_Verde AND Sensor_Succao_Verde AND (Eixo_Z_Verde = REAL#1000) THEN
    etapas_integração := int#13;
END_IF;
(* Rung 12 *)
IF (int#12 = etapas_integração) AND Succao_Azul AND Sensor_Succao_Azul AND (Eixo_Z_Azul = REAL#1000) THEN
    etapas_integração := int#14;
END_IF;
(* Rung 13 *)
IF (int#13 = etapas_integração) AND (Sensor_Z_Verde = REAL#0) THEN etapas_integração := int#15; END_IF;
(* Rung 14 *)
IF (int#14 = etapas_integração) AND (Sensor_Z_Azul = REAL#0) THEN etapas_integração := int#16; END_IF;
(* Rung 15 *)
IF (int#15 = etapas_integração) AND (Sensor_X_Verde = REAL#999) AND NOT Sensor_Rodar_Verde THEN
    etapas_integração := int#17;
END_IF;
(* Rung 16 *)
IF (int#16 = etapas_integração) AND (Sensor_X_Azul = REAL#999) AND NOT Sensor_Rodar_Azul THEN
    etapas_integração := int#18;
END_IF;
(* Rung 17 *)
IF (int#17 = etapas_integração) AND NOT Sensor_Succao_Verde THEN etapas_integração := int#19; END_IF;
(* Rung 18 *)
IF (int#18 = etapas_integração) AND NOT Sensor_Succao_Azul THEN etapas_integração := int#20; END_IF;
(* Rung 19 *)
IF (int#19 = etapas_integração) AND Sensor_Rodar_Verde AND (Sensor_X_Verde > REAL#0) THEN
    etapas_integração := int#21;
END_IF;

